Fanuc KAREL source: kb00122.compact.KL

PROGRAM KB00122
%STACKSIZE=65535
%PRIORITY=65535
%NOLOCKGROUP
%ENVIRONMENT FDEV
VAR
P1 : STRING[80]
P2 : INTEGER
BEGIN
P1='A'
P2=1
MOUNT_DEV(P1,P2)
END KB00122
